{attribute 'qualified_only'}
{attribute 'strict'}
TYPE eHighLevelState :
(
	SLEEP,
	READY,
	OPERATIONAL,
	SHUTDOWN
);
END_TYPE

(* stored: Version 1.1.0.1, ProductVersion 3.1.4024.12
   DUT eHighLevelState: Id {2feee283-07ee-4d6c-9c1d-1916b946fef8} *)
